FUNCTION Convert_DATE_TO_DATE : BOOL
VAR_INPUT
	in : DATE;
	out : REFERENCE TO DATE;
END_VAR

out := in;
Convert_DATE_TO_DATE := TRUE;

END_FUNCTION

(* stored: Version 1.1.0.1, ProductVersion 3.1.4024.12
   POU Convert_DATE_TO_DATE: Id {b6d8be31-60a3-4022-bfa2-36b2288cf930}, SpecialFunc None *)
